// TIA Portal V20 export
FUNCTION_BLOCK "EventsPFE_Recipe"   // FB129, LAD
// stored: MemoryReserve 100, Namespace Unit1.Em11, SetENOAutomatically false
   VAR
      data : Array[1..100] of LReal;
   END_VAR
BEGIN

REGION Network 1: PDR Data61 Recipe - Weight Min Value
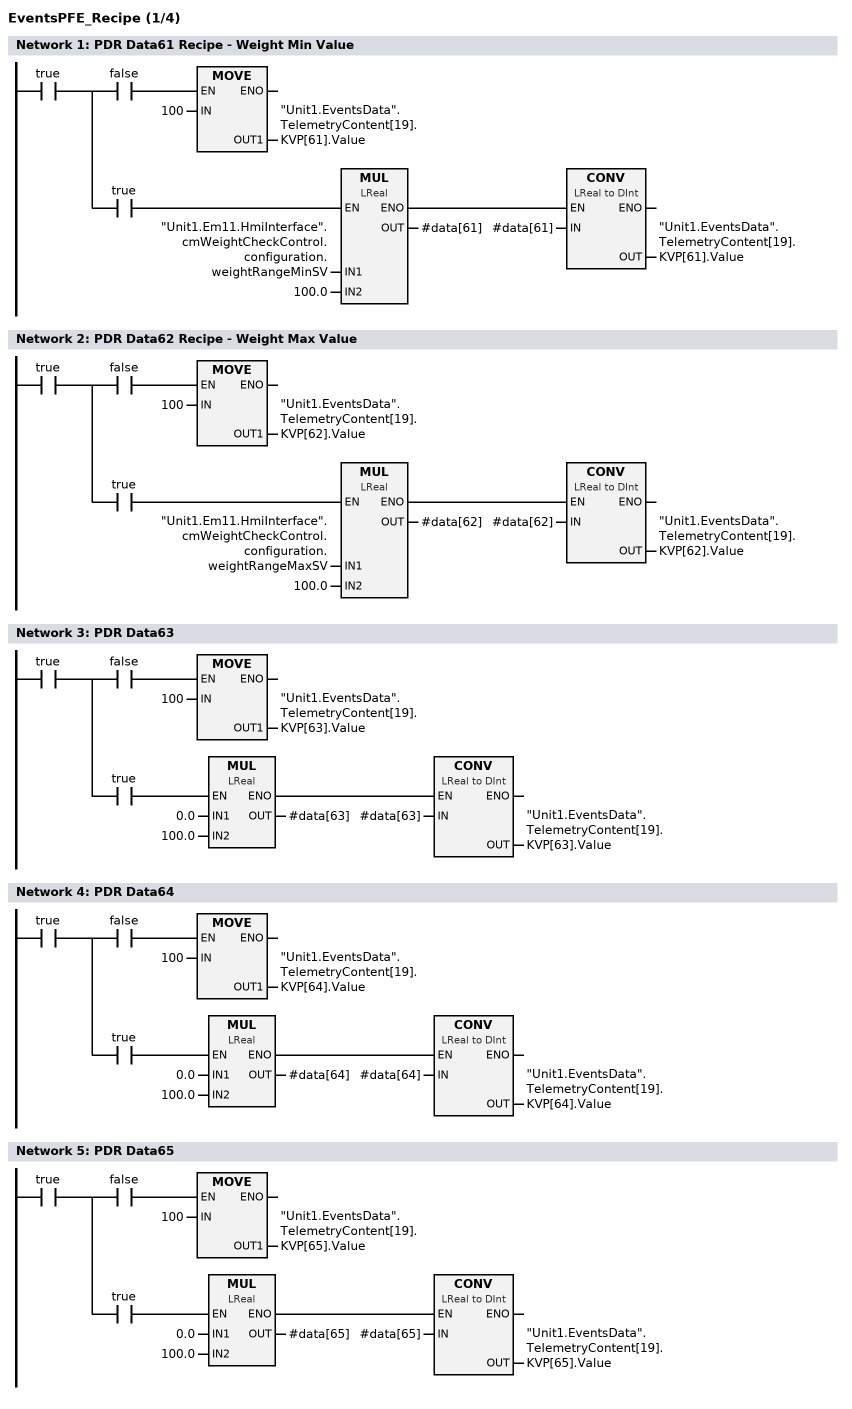
   RUNG wire#powerrail
      Contact( true )
      wire#w1
      Contact( false )
      Move(in := 100, out1 => "Unit1.EventsData".TelemetryContent[19].KVP[61].Value)
   END_RUNG
   RUNG wire#w1
      Contact( true )
      { S7_Templates := "SrcType := LReal" } Mul(in1 := "Unit1.Em11.HmiInterface".cmWeightCheckControl.configuration.weightRangeMinSV, in2 := 100.0, out => #data[61])
      { S7_Templates := "[SrcType := LReal, DestType := DInt]" } Convert(in := #data[61], out => "Unit1.EventsData".TelemetryContent[19].KVP[61].Value)
   END_RUNG
   // the same network as SCL:
   IF true AND false THEN "Unit1.EventsData".TelemetryContent[19].KVP[61].Value := 100; END_IF;
   IF true AND true THEN
       #data[61] := "Unit1.Em11.HmiInterface".cmWeightCheckControl.configuration.weightRangeMinSV * 100.0;
       "Unit1.EventsData".TelemetryContent[19].KVP[61].Value := LREAL_TO_DINT(#data[61]);
   END_IF;
END_REGION

REGION Network 2: PDR Data62 Recipe - Weight Max Value
   RUNG wire#powerrail
      Contact( true )
      wire#w1
      Contact( false )
      Move(in := 100, out1 => "Unit1.EventsData".TelemetryContent[19].KVP[62].Value)
   END_RUNG
   RUNG wire#w1
      Contact( true )
      { S7_Templates := "SrcType := LReal" } Mul(in1 := "Unit1.Em11.HmiInterface".cmWeightCheckControl.configuration.weightRangeMaxSV, in2 := 100.0, out => #data[62])
      { S7_Templates := "[SrcType := LReal, DestType := DInt]" } Convert(in := #data[62], out => "Unit1.EventsData".TelemetryContent[19].KVP[62].Value)
   END_RUNG
   // the same network as SCL:
   IF true AND false THEN "Unit1.EventsData".TelemetryContent[19].KVP[62].Value := 100; END_IF;
   IF true AND true THEN
       #data[62] := "Unit1.Em11.HmiInterface".cmWeightCheckControl.configuration.weightRangeMaxSV * 100.0;
       "Unit1.EventsData".TelemetryContent[19].KVP[62].Value := LREAL_TO_DINT(#data[62]);
   END_IF;
END_REGION

REGION Network 3: PDR Data63
   RUNG wire#powerrail
      Contact( true )
      wire#w1
      Contact( false )
      Move(in := 100, out1 => "Unit1.EventsData".TelemetryContent[19].KVP[63].Value)
   END_RUNG
   RUNG wire#w1
      Contact( true )
      { S7_Templates := "SrcType := LReal" } Mul(in1 := 0.0, in2 := 100.0, out => #data[63])
      { S7_Templates := "[SrcType := LReal, DestType := DInt]" } Convert(in := #data[63], out => "Unit1.EventsData".TelemetryContent[19].KVP[63].Value)
   END_RUNG
   // the same network as SCL:
   IF true AND false THEN "Unit1.EventsData".TelemetryContent[19].KVP[63].Value := 100; END_IF;
   IF true AND true THEN
       #data[63] := 0.0 * 100.0;
       "Unit1.EventsData".TelemetryContent[19].KVP[63].Value := LREAL_TO_DINT(#data[63]);
   END_IF;
END_REGION

REGION Network 4: PDR Data64
   RUNG wire#powerrail
      Contact( true )
      wire#w1
      Contact( false )
      Move(in := 100, out1 => "Unit1.EventsData".TelemetryContent[19].KVP[64].Value)
   END_RUNG
   RUNG wire#w1
      Contact( true )
      { S7_Templates := "SrcType := LReal" } Mul(in1 := 0.0, in2 := 100.0, out => #data[64])
      { S7_Templates := "[SrcType := LReal, DestType := DInt]" } Convert(in := #data[64], out => "Unit1.EventsData".TelemetryContent[19].KVP[64].Value)
   END_RUNG
   // the same network as SCL:
   IF true AND false THEN "Unit1.EventsData".TelemetryContent[19].KVP[64].Value := 100; END_IF;
   IF true AND true THEN
       #data[64] := 0.0 * 100.0;
       "Unit1.EventsData".TelemetryContent[19].KVP[64].Value := LREAL_TO_DINT(#data[64]);
   END_IF;
END_REGION

REGION Network 5: PDR Data65
   RUNG wire#powerrail
      Contact( true )
      wire#w1
      Contact( false )
      Move(in := 100, out1 => "Unit1.EventsData".TelemetryContent[19].KVP[65].Value)
   END_RUNG
   RUNG wire#w1
      Contact( true )
      { S7_Templates := "SrcType := LReal" } Mul(in1 := 0.0, in2 := 100.0, out => #data[65])
      { S7_Templates := "[SrcType := LReal, DestType := DInt]" } Convert(in := #data[65], out => "Unit1.EventsData".TelemetryContent[19].KVP[65].Value)
   END_RUNG
   // the same network as SCL:
   IF true AND false THEN "Unit1.EventsData".TelemetryContent[19].KVP[65].Value := 100; END_IF;
   IF true AND true THEN
       #data[65] := 0.0 * 100.0;
       "Unit1.EventsData".TelemetryContent[19].KVP[65].Value := LREAL_TO_DINT(#data[65]);
   END_IF;
END_REGION

REGION Network 6: PDR Data66
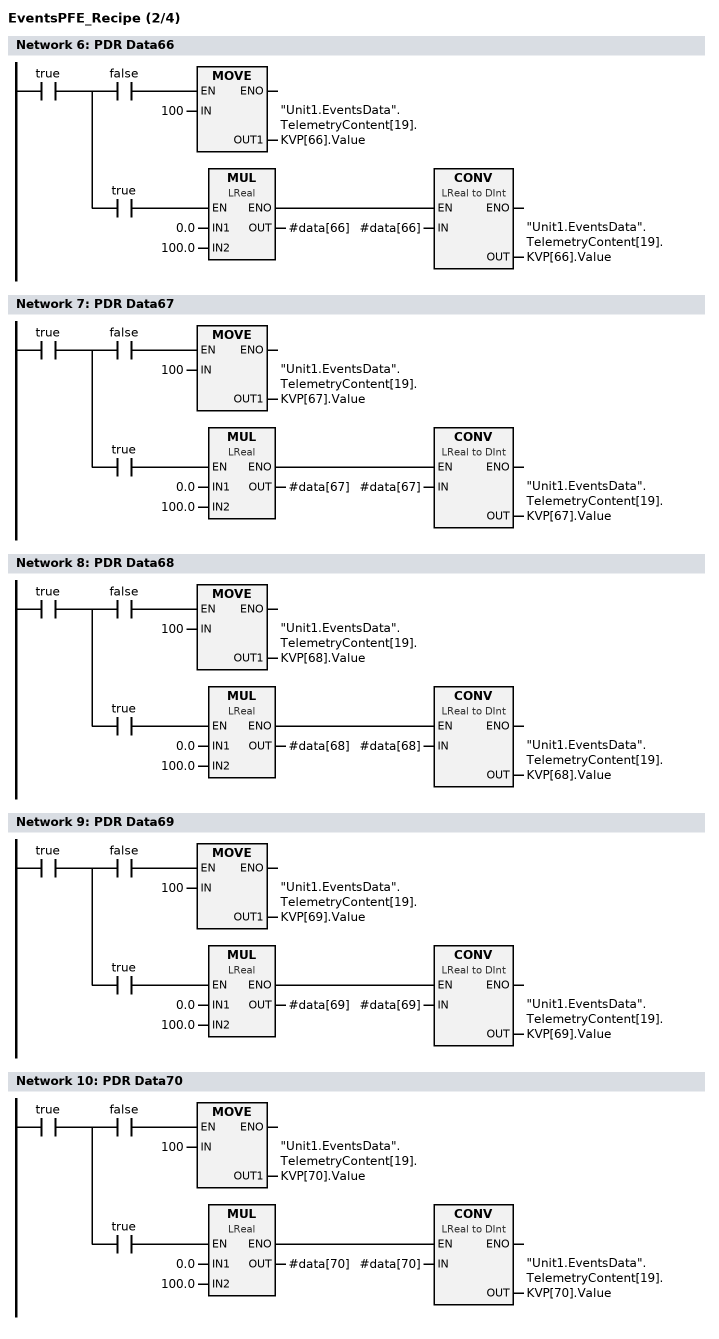
   RUNG wire#powerrail
      Contact( true )
      wire#w1
      Contact( false )
      Move(in := 100, out1 => "Unit1.EventsData".TelemetryContent[19].KVP[66].Value)
   END_RUNG
   RUNG wire#w1
      Contact( true )
      { S7_Templates := "SrcType := LReal" } Mul(in1 := 0.0, in2 := 100.0, out => #data[66])
      { S7_Templates := "[SrcType := LReal, DestType := DInt]" } Convert(in := #data[66], out => "Unit1.EventsData".TelemetryContent[19].KVP[66].Value)
   END_RUNG
   // the same network as SCL:
   IF true AND false THEN "Unit1.EventsData".TelemetryContent[19].KVP[66].Value := 100; END_IF;
   IF true AND true THEN
       #data[66] := 0.0 * 100.0;
       "Unit1.EventsData".TelemetryContent[19].KVP[66].Value := LREAL_TO_DINT(#data[66]);
   END_IF;
END_REGION

REGION Network 7: PDR Data67
   RUNG wire#powerrail
      Contact( true )
      wire#w1
      Contact( false )
      Move(in := 100, out1 => "Unit1.EventsData".TelemetryContent[19].KVP[67].Value)
   END_RUNG
   RUNG wire#w1
      Contact( true )
      { S7_Templates := "SrcType := LReal" } Mul(in1 := 0.0, in2 := 100.0, out => #data[67])
      { S7_Templates := "[SrcType := LReal, DestType := DInt]" } Convert(in := #data[67], out => "Unit1.EventsData".TelemetryContent[19].KVP[67].Value)
   END_RUNG
   // the same network as SCL:
   IF true AND false THEN "Unit1.EventsData".TelemetryContent[19].KVP[67].Value := 100; END_IF;
   IF true AND true THEN
       #data[67] := 0.0 * 100.0;
       "Unit1.EventsData".TelemetryContent[19].KVP[67].Value := LREAL_TO_DINT(#data[67]);
   END_IF;
END_REGION

REGION Network 8: PDR Data68
   RUNG wire#powerrail
      Contact( true )
      wire#w1
      Contact( false )
      Move(in := 100, out1 => "Unit1.EventsData".TelemetryContent[19].KVP[68].Value)
   END_RUNG
   RUNG wire#w1
      Contact( true )
      { S7_Templates := "SrcType := LReal" } Mul(in1 := 0.0, in2 := 100.0, out => #data[68])
      { S7_Templates := "[SrcType := LReal, DestType := DInt]" } Convert(in := #data[68], out => "Unit1.EventsData".TelemetryContent[19].KVP[68].Value)
   END_RUNG
   // the same network as SCL:
   IF true AND false THEN "Unit1.EventsData".TelemetryContent[19].KVP[68].Value := 100; END_IF;
   IF true AND true THEN
       #data[68] := 0.0 * 100.0;
       "Unit1.EventsData".TelemetryContent[19].KVP[68].Value := LREAL_TO_DINT(#data[68]);
   END_IF;
END_REGION

REGION Network 9: PDR Data69
   RUNG wire#powerrail
      Contact( true )
      wire#w1
      Contact( false )
      Move(in := 100, out1 => "Unit1.EventsData".TelemetryContent[19].KVP[69].Value)
   END_RUNG
   RUNG wire#w1
      Contact( true )
      { S7_Templates := "SrcType := LReal" } Mul(in1 := 0.0, in2 := 100.0, out => #data[69])
      { S7_Templates := "[SrcType := LReal, DestType := DInt]" } Convert(in := #data[69], out => "Unit1.EventsData".TelemetryContent[19].KVP[69].Value)
   END_RUNG
   // the same network as SCL:
   IF true AND false THEN "Unit1.EventsData".TelemetryContent[19].KVP[69].Value := 100; END_IF;
   IF true AND true THEN
       #data[69] := 0.0 * 100.0;
       "Unit1.EventsData".TelemetryContent[19].KVP[69].Value := LREAL_TO_DINT(#data[69]);
   END_IF;
END_REGION

REGION Network 10: PDR Data70
   RUNG wire#powerrail
      Contact( true )
      wire#w1
      Contact( false )
      Move(in := 100, out1 => "Unit1.EventsData".TelemetryContent[19].KVP[70].Value)
   END_RUNG
   RUNG wire#w1
      Contact( true )
      { S7_Templates := "SrcType := LReal" } Mul(in1 := 0.0, in2 := 100.0, out => #data[70])
      { S7_Templates := "[SrcType := LReal, DestType := DInt]" } Convert(in := #data[70], out => "Unit1.EventsData".TelemetryContent[19].KVP[70].Value)
   END_RUNG
   // the same network as SCL:
   IF true AND false THEN "Unit1.EventsData".TelemetryContent[19].KVP[70].Value := 100; END_IF;
   IF true AND true THEN
       #data[70] := 0.0 * 100.0;
       "Unit1.EventsData".TelemetryContent[19].KVP[70].Value := LREAL_TO_DINT(#data[70]);
   END_IF;
END_REGION

REGION Network 11: PDR Data71
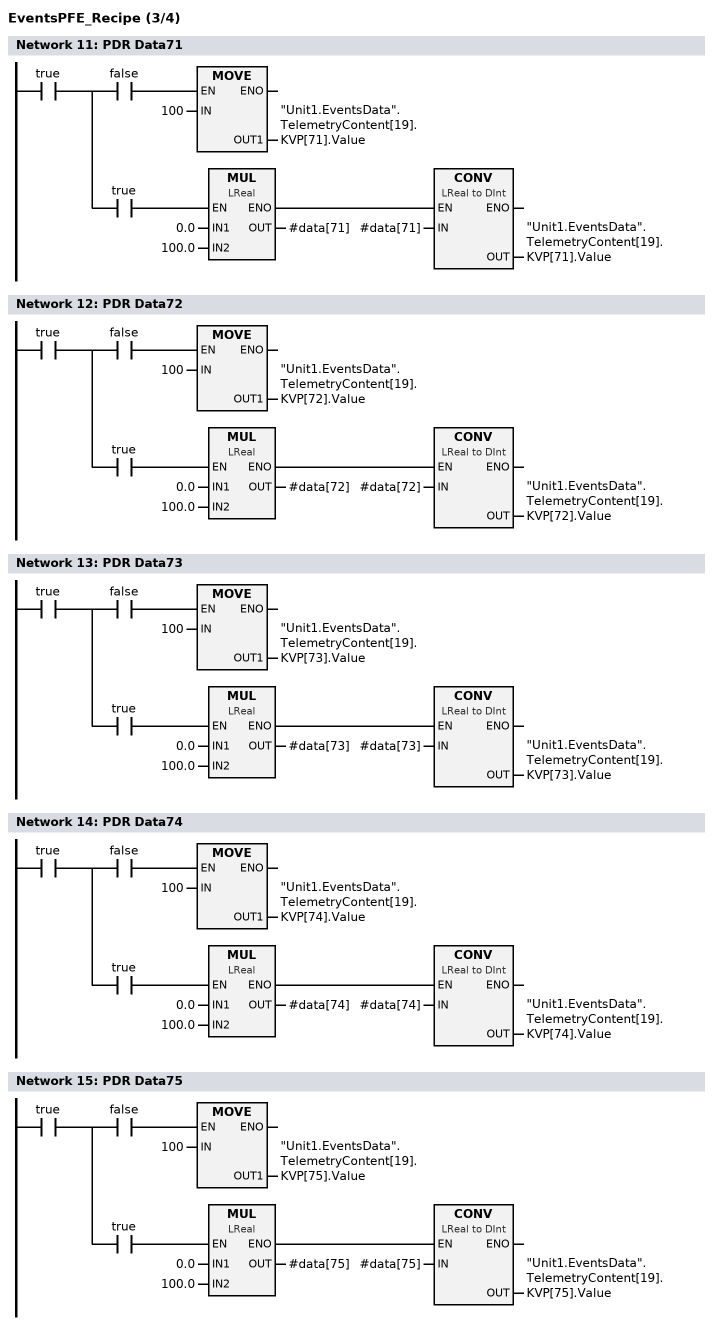
   RUNG wire#powerrail
      Contact( true )
      wire#w1
      Contact( false )
      Move(in := 100, out1 => "Unit1.EventsData".TelemetryContent[19].KVP[71].Value)
   END_RUNG
   RUNG wire#w1
      Contact( true )
      { S7_Templates := "SrcType := LReal" } Mul(in1 := 0.0, in2 := 100.0, out => #data[71])
      { S7_Templates := "[SrcType := LReal, DestType := DInt]" } Convert(in := #data[71], out => "Unit1.EventsData".TelemetryContent[19].KVP[71].Value)
   END_RUNG
   // the same network as SCL:
   IF true AND false THEN "Unit1.EventsData".TelemetryContent[19].KVP[71].Value := 100; END_IF;
   IF true AND true THEN
       #data[71] := 0.0 * 100.0;
       "Unit1.EventsData".TelemetryContent[19].KVP[71].Value := LREAL_TO_DINT(#data[71]);
   END_IF;
END_REGION

REGION Network 12: PDR Data72
   RUNG wire#powerrail
      Contact( true )
      wire#w1
      Contact( false )
      Move(in := 100, out1 => "Unit1.EventsData".TelemetryContent[19].KVP[72].Value)
   END_RUNG
   RUNG wire#w1
      Contact( true )
      { S7_Templates := "SrcType := LReal" } Mul(in1 := 0.0, in2 := 100.0, out => #data[72])
      { S7_Templates := "[SrcType := LReal, DestType := DInt]" } Convert(in := #data[72], out => "Unit1.EventsData".TelemetryContent[19].KVP[72].Value)
   END_RUNG
   // the same network as SCL:
   IF true AND false THEN "Unit1.EventsData".TelemetryContent[19].KVP[72].Value := 100; END_IF;
   IF true AND true THEN
       #data[72] := 0.0 * 100.0;
       "Unit1.EventsData".TelemetryContent[19].KVP[72].Value := LREAL_TO_DINT(#data[72]);
   END_IF;
END_REGION

REGION Network 13: PDR Data73
   RUNG wire#powerrail
      Contact( true )
      wire#w1
      Contact( false )
      Move(in := 100, out1 => "Unit1.EventsData".TelemetryContent[19].KVP[73].Value)
   END_RUNG
   RUNG wire#w1
      Contact( true )
      { S7_Templates := "SrcType := LReal" } Mul(in1 := 0.0, in2 := 100.0, out => #data[73])
      { S7_Templates := "[SrcType := LReal, DestType := DInt]" } Convert(in := #data[73], out => "Unit1.EventsData".TelemetryContent[19].KVP[73].Value)
   END_RUNG
   // the same network as SCL:
   IF true AND false THEN "Unit1.EventsData".TelemetryContent[19].KVP[73].Value := 100; END_IF;
   IF true AND true THEN
       #data[73] := 0.0 * 100.0;
       "Unit1.EventsData".TelemetryContent[19].KVP[73].Value := LREAL_TO_DINT(#data[73]);
   END_IF;
END_REGION

REGION Network 14: PDR Data74
   RUNG wire#powerrail
      Contact( true )
      wire#w1
      Contact( false )
      Move(in := 100, out1 => "Unit1.EventsData".TelemetryContent[19].KVP[74].Value)
   END_RUNG
   RUNG wire#w1
      Contact( true )
      { S7_Templates := "SrcType := LReal" } Mul(in1 := 0.0, in2 := 100.0, out => #data[74])
      { S7_Templates := "[SrcType := LReal, DestType := DInt]" } Convert(in := #data[74], out => "Unit1.EventsData".TelemetryContent[19].KVP[74].Value)
   END_RUNG
   // the same network as SCL:
   IF true AND false THEN "Unit1.EventsData".TelemetryContent[19].KVP[74].Value := 100; END_IF;
   IF true AND true THEN
       #data[74] := 0.0 * 100.0;
       "Unit1.EventsData".TelemetryContent[19].KVP[74].Value := LREAL_TO_DINT(#data[74]);
   END_IF;
END_REGION

REGION Network 15: PDR Data75
   RUNG wire#powerrail
      Contact( true )
      wire#w1
      Contact( false )
      Move(in := 100, out1 => "Unit1.EventsData".TelemetryContent[19].KVP[75].Value)
   END_RUNG
   RUNG wire#w1
      Contact( true )
      { S7_Templates := "SrcType := LReal" } Mul(in1 := 0.0, in2 := 100.0, out => #data[75])
      { S7_Templates := "[SrcType := LReal, DestType := DInt]" } Convert(in := #data[75], out => "Unit1.EventsData".TelemetryContent[19].KVP[75].Value)
   END_RUNG
   // the same network as SCL:
   IF true AND false THEN "Unit1.EventsData".TelemetryContent[19].KVP[75].Value := 100; END_IF;
   IF true AND true THEN
       #data[75] := 0.0 * 100.0;
       "Unit1.EventsData".TelemetryContent[19].KVP[75].Value := LREAL_TO_DINT(#data[75]);
   END_IF;
END_REGION

REGION Network 16: PDR Data76
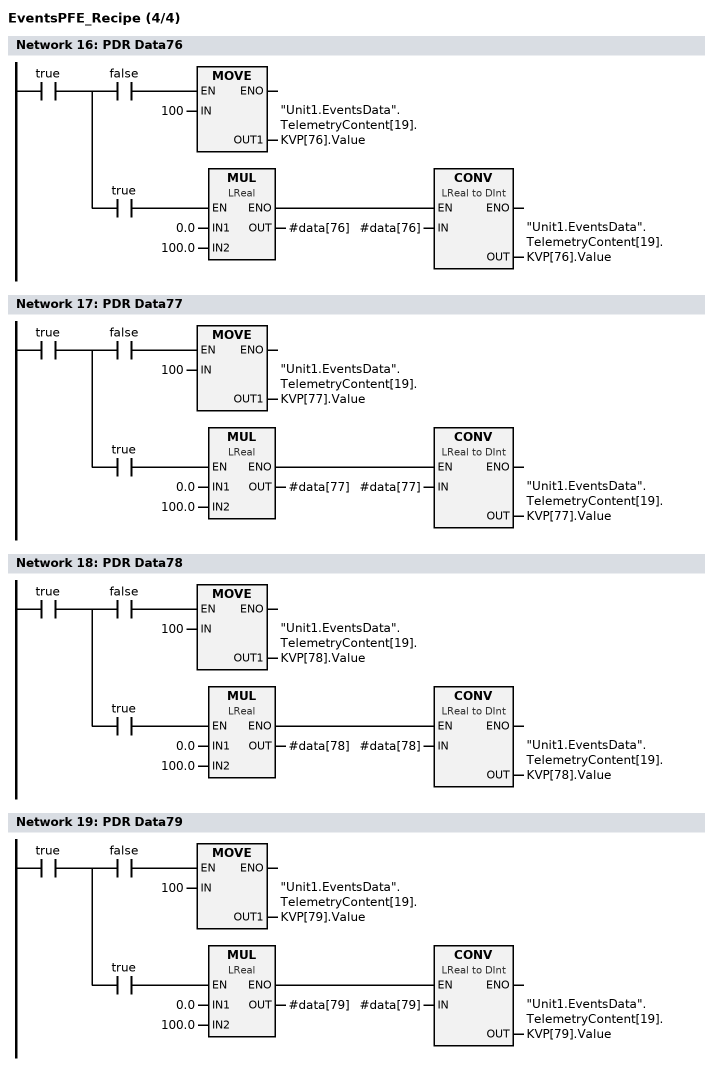
   RUNG wire#powerrail
      Contact( true )
      wire#w1
      Contact( false )
      Move(in := 100, out1 => "Unit1.EventsData".TelemetryContent[19].KVP[76].Value)
   END_RUNG
   RUNG wire#w1
      Contact( true )
      { S7_Templates := "SrcType := LReal" } Mul(in1 := 0.0, in2 := 100.0, out => #data[76])
      { S7_Templates := "[SrcType := LReal, DestType := DInt]" } Convert(in := #data[76], out => "Unit1.EventsData".TelemetryContent[19].KVP[76].Value)
   END_RUNG
   // the same network as SCL:
   IF true AND false THEN "Unit1.EventsData".TelemetryContent[19].KVP[76].Value := 100; END_IF;
   IF true AND true THEN
       #data[76] := 0.0 * 100.0;
       "Unit1.EventsData".TelemetryContent[19].KVP[76].Value := LREAL_TO_DINT(#data[76]);
   END_IF;
END_REGION

REGION Network 17: PDR Data77
   RUNG wire#powerrail
      Contact( true )
      wire#w1
      Contact( false )
      Move(in := 100, out1 => "Unit1.EventsData".TelemetryContent[19].KVP[77].Value)
   END_RUNG
   RUNG wire#w1
      Contact( true )
      { S7_Templates := "SrcType := LReal" } Mul(in1 := 0.0, in2 := 100.0, out => #data[77])
      { S7_Templates := "[SrcType := LReal, DestType := DInt]" } Convert(in := #data[77], out => "Unit1.EventsData".TelemetryContent[19].KVP[77].Value)
   END_RUNG
   // the same network as SCL:
   IF true AND false THEN "Unit1.EventsData".TelemetryContent[19].KVP[77].Value := 100; END_IF;
   IF true AND true THEN
       #data[77] := 0.0 * 100.0;
       "Unit1.EventsData".TelemetryContent[19].KVP[77].Value := LREAL_TO_DINT(#data[77]);
   END_IF;
END_REGION

REGION Network 18: PDR Data78
   RUNG wire#powerrail
      Contact( true )
      wire#w1
      Contact( false )
      Move(in := 100, out1 => "Unit1.EventsData".TelemetryContent[19].KVP[78].Value)
   END_RUNG
   RUNG wire#w1
      Contact( true )
      { S7_Templates := "SrcType := LReal" } Mul(in1 := 0.0, in2 := 100.0, out => #data[78])
      { S7_Templates := "[SrcType := LReal, DestType := DInt]" } Convert(in := #data[78], out => "Unit1.EventsData".TelemetryContent[19].KVP[78].Value)
   END_RUNG
   // the same network as SCL:
   IF true AND false THEN "Unit1.EventsData".TelemetryContent[19].KVP[78].Value := 100; END_IF;
   IF true AND true THEN
       #data[78] := 0.0 * 100.0;
       "Unit1.EventsData".TelemetryContent[19].KVP[78].Value := LREAL_TO_DINT(#data[78]);
   END_IF;
END_REGION

REGION Network 19: PDR Data79
   RUNG wire#powerrail
      Contact( true )
      wire#w1
      Contact( false )
      Move(in := 100, out1 => "Unit1.EventsData".TelemetryContent[19].KVP[79].Value)
   END_RUNG
   RUNG wire#w1
      Contact( true )
      { S7_Templates := "SrcType := LReal" } Mul(in1 := 0.0, in2 := 100.0, out => #data[79])
      { S7_Templates := "[SrcType := LReal, DestType := DInt]" } Convert(in := #data[79], out => "Unit1.EventsData".TelemetryContent[19].KVP[79].Value)
   END_RUNG
   // the same network as SCL:
   IF true AND false THEN "Unit1.EventsData".TelemetryContent[19].KVP[79].Value := 100; END_IF;
   IF true AND true THEN
       #data[79] := 0.0 * 100.0;
       "Unit1.EventsData".TelemetryContent[19].KVP[79].Value := LREAL_TO_DINT(#data[79]);
   END_IF;
END_REGION
END_FUNCTION_BLOCK
